# EPICS autosave request: iocBoot/generic_motors_ioc/dbSave/bluiceScan.req
$(P)edgeEnergy
$(P)edgeCutoff
$(P)time
$(P)roiLow
$(P)roiHigh
$(P)adcGain
$(P)adcOffset
$(P)optADCGain
$(P)optADCOffset
$(P)startScan
$(P)stopScan
$(P)endScan
